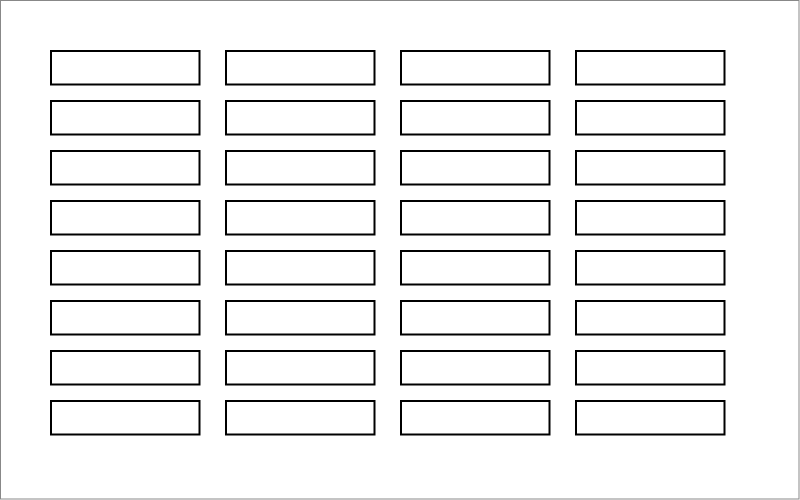
VISUALIZATION Screen_1_Sub_3  // 800x500
    Rectangle (50,50 150x35), "Val 1: %i", text variable: GVL.HMI_Display_Int[0]
    Rectangle (225,50 150x35), "Val 2: %i", text variable: GVL.HMI_Display_Int[1]
    Rectangle (400,50 150x35), "Val 3: %i", text variable: GVL.HMI_Display_Int[2]
    Rectangle (575,50 150x35), "Val 4: %i", text variable: GVL.HMI_Display_Int[3]
    Rectangle (50,100 150x35), "Val 5: %i", text variable: GVL.HMI_Display_Int[4]
    Rectangle (225,100 150x35), "Val 6: %i", text variable: GVL.HMI_Display_Int[5]
    Rectangle (400,100 150x35), "Val 7: %i", text variable: GVL.HMI_Display_Int[6]
    Rectangle (575,100 150x35), "Val 8: %i", text variable: GVL.HMI_Display_Int[7]
    Rectangle (50,150 150x35), "Val 9: %i", text variable: GVL.HMI_Display_Int[8]
    Rectangle (225,150 150x35), "Val 10: %i", text variable: GVL.HMI_Display_Int[9]
    Rectangle (400,150 150x35), "Val 11: %i", text variable: GVL.HMI_Display_Int[10]
    Rectangle (575,150 150x35), "Val 12: %i", text variable: GVL.HMI_Display_Int[11]
    Rectangle (50,200 150x35), "Val 13: %i", text variable: GVL.HMI_Display_Int[12]
    Rectangle (225,200 150x35), "Val 14: %i", text variable: GVL.HMI_Display_Int[13]
    Rectangle (400,200 150x35), "Val 15: %i", text variable: GVL.HMI_Display_Int[14]
    Rectangle (575,200 150x35), "Val 16: %i", text variable: GVL.HMI_Display_Int[15]
    Rectangle (50,250 150x35), "Val 17: %i", text variable: GVL.HMI_Display_Int[16]
    Rectangle (225,250 150x35), "Val 18: %i", text variable: GVL.HMI_Display_Int[17]
    Rectangle (400,250 150x35), "Val 19: %i", text variable: GVL.HMI_Display_Int[18]
    Rectangle (575,250 150x35), "Val 20: %i", text variable: GVL.HMI_Display_Int[19]
    Rectangle (50,300 150x35), "Val 21: %i", text variable: GVL.HMI_Display_Int[20]
    Rectangle (225,300 150x35), "Val 22: %i", text variable: GVL.HMI_Display_Int[21]
    Rectangle (400,300 150x35), "Val 23: %i", text variable: GVL.HMI_Display_Int[22]
    Rectangle (575,300 150x35), "Val 24: %i", text variable: GVL.HMI_Display_Int[23]
    Rectangle (50,350 150x35), "Val 25: %i", text variable: GVL.HMI_Display_Int[24]
    Rectangle (225,350 150x35), "Val 26: %i", text variable: GVL.HMI_Display_Int[25]
    Rectangle (400,350 150x35), "Val 27: %i", text variable: GVL.HMI_Display_Int[26]
    Rectangle (575,350 150x35), "Val 28: %i", text variable: GVL.HMI_Display_Int[27]
    Rectangle (50,400 150x35), "Val 29: %i", text variable: GVL.HMI_Display_Int[28]
    Rectangle (225,400 150x35), "Val 30: %i", text variable: GVL.HMI_Display_Int[29]
    Rectangle (400,400 150x35), "Val 31: %i", text variable: GVL.HMI_Display_Int[30]
    Rectangle (575,400 150x35), "Val 32: %i", text variable: GVL.HMI_Display_Int[31]
END_VISUALIZATION

(* stored: Version 1.1.0.1, ProductVersion 3.1.4024.12
   Visu Screen_1_Sub_3: Id {d116871a-d098-4a66-ae61-4d315a7491ed} *)
